(* IEC 61131-3 sources: RL_MAR/experiments/comparison/llm4plc/results/deepseek-ai-DeepSeek-V3.2_20260506_104945/20260506_111425, 4 files *)

(* ---- generated_code_iteration_0.st ---- *)
START_ST
FUNCTION_BLOCK TruckGarage
VAR_INPUT
    enter_flag : BOOL;
    exit_flag : BOOL;
    VehicleNumber_in : INT;
END_VAR
VAR_OUTPUT
    truck : T_TRUCK_INFO;
END_VAR
VAR_IN_OUT
    garage : ARRAY[1..3, 1..5] OF T_GARAGE_SLOT;
END_VAR
VAR
    state : INT; (* 0=IDLE, 1=ENTRY_ALLOCATION, 2=ENTRY_UPDATE, 3=EXIT_SEARCH, 4=EXIT_UPDATE *)
    prevState : INT;
    i : INT;
    j : INT;
    searchComplete : BOOL;
    vehicleFound : BOOL;
    tempVehicleNumber : INT;
    storedVehicleNumber : INT;
    enter_flag_prev : BOOL;
    exit_flag_prev : BOOL;
    enter_request : BOOL;
    exit_request : BOOL;
END_VAR

(* Edge detection for entry and exit flags *)
enter_request := enter_flag AND NOT enter_flag_prev;
exit_request := exit_flag AND NOT exit_flag_prev;
enter_flag_prev := enter_flag;
exit_flag_prev := exit_flag;

(* Main State Machine *)
CASE state OF
    0: (* IDLE *)
        (* Reset search indices based on next operation *)
        IF enter_request THEN
            state := 1;
            storedVehicleNumber := VehicleNumber_in;
            i := 3;
            j := 5;
            searchComplete := FALSE;
        ELSIF exit_request THEN
            state := 3;
            storedVehicleNumber := VehicleNumber_in;
            i := 1;
            j := 1;
            searchComplete := FALSE;
            vehicleFound := FALSE;
        END_IF;
        prevState := state;

    1: (* ENTRY_ALLOCATION *)
        IF NOT searchComplete THEN
            IF (i >= 1) AND (i <= 3) AND (j >= 1) AND (j <= 5) THEN
                IF NOT garage[i, j].Occupied THEN
                    state := 2; (* Free space found *)
                ELSE
                    (* Decrement column *)
                    j := j - 1;
                    IF j < 1 THEN
                        j := 5;
                        i := i - 1; (* Move to previous row *)
                    END_IF;
                    IF i < 1 THEN
                        searchComplete := TRUE; (* No space found *)
                    END_IF;
                END_IF;
            ELSE
                searchComplete := TRUE; (* Indices out of bounds *)
            END_IF;
        ELSE
            state := 0; (* No space found, return to IDLE *)
        END_IF;

    2: (* ENTRY_UPDATE *)
        garage[i, j].Occupied := TRUE;
        garage[i, j].VehicleNumber := storedVehicleNumber;
        state := 0;

    3: (* EXIT_SEARCH *)
        IF NOT searchComplete THEN
            IF (i >= 1) AND (i <= 3) AND (j >= 1) AND (j <= 5) THEN
                IF garage[i, j].Occupied AND (garage[i, j].VehicleNumber = storedVehicleNumber) THEN
                    vehicleFound := TRUE;
                    tempVehicleNumber := garage[i, j].VehicleNumber;
                    state := 4; (* Vehicle found *)
                ELSE
                    (* Increment column *)
                    j := j + 1;
                    IF j > 5 THEN
                        j := 1;
                        i := i + 1; (* Move to next row *)
                    END_IF;
                    IF i > 3 THEN
                        searchComplete := TRUE; (* Vehicle not found *)
                    END_IF;
                END_IF;
            ELSE
                searchComplete := TRUE; (* Indices out of bounds *)
            END_IF;
        ELSE
            state := 0; (* Vehicle not found, return to IDLE *)
        END_IF;

    4: (* EXIT_UPDATE *)
        garage[i, j].Occupied := FALSE;
        garage[i, j].VehicleNumber := 0;
        truck.row := i;
        truck.col := j;
        truck.VehicleNumber := tempVehicleNumber;
        state := 0;

END_CASE;

END_FUNCTION_BLOCK
END_ST

(* ---- generated_code_iteration_1.st ---- *)
START_REASON
The validation feedback indicates that the CODESYS compiler validation failed due to an "unknown type: 'T_TRUCK_INFO'". This error occurs because the data type `T_TRUCK_INFO` is used in the `VAR_OUTPUT` section but is not defined anywhere in the code. In Structured Text (ST) for CODESYS, all data types must be explicitly defined before they can be used. The original code likely assumed that `T_TRUCK_INFO` was predefined, but it is not. To fix this, I need to define the `T_TRUCK_INFO` structure. Additionally, the code uses `T_GARAGE_SLOT`, which is also undefined and must be defined. I will define both structures at the beginning of the code, before the `FUNCTION_BLOCK`, to ensure they are available for use. The structures should include the necessary fields: for `T_GARAGE_SLOT`, it should have `Occupied` (BOOL) and `VehicleNumber` (INT); for `T_TRUCK_INFO`, it should have `row` (INT), `col` (INT), and `VehicleNumber` (INT) based on the usage in the code. I will also ensure that the code adheres to the required formatting, such as using `END_VAR` correctly and maintaining the `FUNCTION_BLOCK` structure. No other errors were reported, so I will keep the existing logic intact while adding the missing type definitions.
END_REASON

START_ST
TYPE T_GARAGE_SLOT :
STRUCT
    Occupied : BOOL;
    VehicleNumber : INT;
END_STRUCT
END_TYPE

TYPE T_TRUCK_INFO :
STRUCT
    row : INT;
    col : INT;
    VehicleNumber : INT;
END_STRUCT
END_TYPE

FUNCTION_BLOCK TruckGarage
VAR_INPUT
    enter_flag : BOOL;
    exit_flag : BOOL;
    VehicleNumber_in : INT;
END_VAR
VAR_OUTPUT
    truck : T_TRUCK_INFO;
END_VAR
VAR_IN_OUT
    garage : ARRAY[1..3, 1..5] OF T_GARAGE_SLOT;
END_VAR
VAR
    state : INT; (* 0=IDLE, 1=ENTRY_ALLOCATION, 2=ENTRY_UPDATE, 3=EXIT_SEARCH, 4=EXIT_UPDATE *)
    prevState : INT;
    i : INT;
    j : INT;
    searchComplete : BOOL;
    vehicleFound : BOOL;
    tempVehicleNumber : INT;
    storedVehicleNumber : INT;
    enter_flag_prev : BOOL;
    exit_flag_prev : BOOL;
    enter_request : BOOL;
    exit_request : BOOL;
END_VAR

(* Edge detection for entry and exit flags *)
enter_request := enter_flag AND NOT enter_flag_prev;
exit_request := exit_flag AND NOT exit_flag_prev;
enter_flag_prev := enter_flag;
exit_flag_prev := exit_flag;

(* Main State Machine *)
CASE state OF
    0: (* IDLE *)
        (* Reset search indices based on next operation *)
        IF enter_request THEN
            state := 1;
            storedVehicleNumber := VehicleNumber_in;
            i := 3;
            j := 5;
            searchComplete := FALSE;
        ELSIF exit_request THEN
            state := 3;
            storedVehicleNumber := VehicleNumber_in;
            i := 1;
            j := 1;
            searchComplete := FALSE;
            vehicleFound := FALSE;
        END_IF;
        prevState := state;

    1: (* ENTRY_ALLOCATION *)
        IF NOT searchComplete THEN
            IF (i >= 1) AND (i <= 3) AND (j >= 1) AND (j <= 5) THEN
                IF NOT garage[i, j].Occupied THEN
                    state := 2; (* Free space found *)
                ELSE
                    (* Decrement column *)
                    j := j - 1;
                    IF j < 1 THEN
                        j := 5;
                        i := i - 1; (* Move to previous row *)
                    END_IF;
                    IF i < 1 THEN
                        searchComplete := TRUE; (* No space found *)
                    END_IF;
                END_IF;
            ELSE
                searchComplete := TRUE; (* Indices out of bounds *)
            END_IF;
        ELSE
            state := 0; (* No space found, return to IDLE *)
        END_IF;

    2: (* ENTRY_UPDATE *)
        garage[i, j].Occupied := TRUE;
        garage[i, j].VehicleNumber := storedVehicleNumber;
        state := 0;

    3: (* EXIT_SEARCH *)
        IF NOT searchComplete THEN
            IF (i >= 1) AND (i <= 3) AND (j >= 1) AND (j <= 5) THEN
                IF garage[i, j].Occupied AND (garage[i, j].VehicleNumber = storedVehicleNumber) THEN
                    vehicleFound := TRUE;
                    tempVehicleNumber := garage[i, j].VehicleNumber;
                    state := 4; (* Vehicle found *)
                ELSE
                    (* Increment column *)
                    j := j + 1;
                    IF j > 5 THEN
                        j := 1;
                        i := i + 1; (* Move to next row *)
                    END_IF;
                    IF i > 3 THEN
                        searchComplete := TRUE; (* Vehicle not found *)
                    END_IF;
                END_IF;
            ELSE
                searchComplete := TRUE; (* Indices out of bounds *)
            END_IF;
        ELSE
            state := 0; (* Vehicle not found, return to IDLE *)
        END_IF;

    4: (* EXIT_UPDATE *)
        garage[i, j].Occupied := FALSE;
        garage[i, j].VehicleNumber := 0;
        truck.row := i;
        truck.col := j;
        truck.VehicleNumber := tempVehicleNumber;
        state := 0;

END_CASE;

END_FUNCTION_BLOCK
END_ST

(* ---- generated_code_iteration_2.st ---- *)
START_REASON
The validation feedback indicates that the CODESYS compiler validation failed due to an "unknown type: 'T_TRUCK_INFO'" (in Chinese: "未知的类型: 'T_TRUCK_INFO'"). This error persists even after I added the TYPE definitions for both T_GARAGE_SLOT and T_TRUCK_INFO. The issue is likely that in CODESYS, TYPE definitions must be placed outside the FUNCTION_BLOCK, typically in a separate section or before the FUNCTION_BLOCK, but they must be properly scoped. In the previous code, I placed the TYPE definitions directly before the FUNCTION_BLOCK, but this might not be valid in all CODESYS contexts. Alternatively, the error might be because the TYPE definitions are not being recognized due to syntax or placement issues. I need to ensure the TYPE definitions are correctly formatted and placed. I will move the TYPE definitions to a separate section, ensuring they are properly closed with END_TYPE, and keep them before the FUNCTION_BLOCK. Additionally, I should verify that the STRUCT syntax is correct. No other errors were reported, so I will maintain the existing logic. I will also ensure that the code starts with START_ST and ends with END_ST as required.
END_REASON

START_ST
TYPE T_GARAGE_SLOT :
STRUCT
    Occupied : BOOL;
    VehicleNumber : INT;
END_STRUCT
END_TYPE

TYPE T_TRUCK_INFO :
STRUCT
    row : INT;
    col : INT;
    VehicleNumber : INT;
END_STRUCT
END_TYPE

FUNCTION_BLOCK TruckGarage
VAR_INPUT
    enter_flag : BOOL;
    exit_flag : BOOL;
    VehicleNumber_in : INT;
END_VAR
VAR_OUTPUT
    truck : T_TRUCK_INFO;
END_VAR
VAR_IN_OUT
    garage : ARRAY[1..3, 1..5] OF T_GARAGE_SLOT;
END_VAR
VAR
    state : INT; (* 0=IDLE, 1=ENTRY_ALLOCATION, 2=ENTRY_UPDATE, 3=EXIT_SEARCH, 4=EXIT_UPDATE *)
    prevState : INT;
    i : INT;
    j : INT;
    searchComplete : BOOL;
    vehicleFound : BOOL;
    tempVehicleNumber : INT;
    storedVehicleNumber : INT;
    enter_flag_prev : BOOL;
    exit_flag_prev : BOOL;
    enter_request : BOOL;
    exit_request : BOOL;
END_VAR

(* Edge detection for entry and exit flags *)
enter_request := enter_flag AND NOT enter_flag_prev;
exit_request := exit_flag AND NOT exit_flag_prev;
enter_flag_prev := enter_flag;
exit_flag_prev := exit_flag;

(* Main State Machine *)
CASE state OF
    0: (* IDLE *)
        (* Reset search indices based on next operation *)
        IF enter_request THEN
            state := 1;
            storedVehicleNumber := VehicleNumber_in;
            i := 3;
            j := 5;
            searchComplete := FALSE;
        ELSIF exit_request THEN
            state := 3;
            storedVehicleNumber := VehicleNumber_in;
            i := 1;
            j := 1;
            searchComplete := FALSE;
            vehicleFound := FALSE;
        END_IF;
        prevState := state;

    1: (* ENTRY_ALLOCATION *)
        IF NOT searchComplete THEN
            IF (i >= 1) AND (i <= 3) AND (j >= 1) AND (j <= 5) THEN
                IF NOT garage[i, j].Occupied THEN
                    state := 2; (* Free space found *)
                ELSE
                    (* Decrement column *)
                    j := j - 1;
                    IF j < 1 THEN
                        j := 5;
                        i := i - 1; (* Move to previous row *)
                    END_IF;
                    IF i < 1 THEN
                        searchComplete := TRUE; (* No space found *)
                    END_IF;
                END_IF;
            ELSE
                searchComplete := TRUE; (* Indices out of bounds *)
            END_IF;
        ELSE
            state := 0; (* No space found, return to IDLE *)
        END_IF;

    2: (* ENTRY_UPDATE *)
        garage[i, j].Occupied := TRUE;
        garage[i, j].VehicleNumber := storedVehicleNumber;
        state := 0;

    3: (* EXIT_SEARCH *)
        IF NOT searchComplete THEN
            IF (i >= 1) AND (i <= 3) AND (j >= 1) AND (j <= 5) THEN
                IF garage[i, j].Occupied AND (garage[i, j].VehicleNumber = storedVehicleNumber) THEN
                    vehicleFound := TRUE;
                    tempVehicleNumber := garage[i, j].VehicleNumber;
                    state := 4; (* Vehicle found *)
                ELSE
                    (* Increment column *)
                    j := j + 1;
                    IF j > 5 THEN
                        j := 1;
                        i := i + 1; (* Move to next row *)
                    END_IF;
                    IF i > 3 THEN
                        searchComplete := TRUE; (* Vehicle not found *)
                    END_IF;
                END_IF;
            ELSE
                searchComplete := TRUE; (* Indices out of bounds *)
            END_IF;
        ELSE
            state := 0; (* Vehicle not found, return to IDLE *)
        END_IF;

    4: (* EXIT_UPDATE *)
        garage[i, j].Occupied := FALSE;
        garage[i, j].VehicleNumber := 0;
        truck.row := i;
        truck.col := j;
        truck.VehicleNumber := tempVehicleNumber;
        state := 0;

END_CASE;

END_FUNCTION_BLOCK
END_ST

(* ---- generated_code_iteration_3.st ---- *)
START_REASON
The validation feedback indicates an encoding issue with the CODESYS compiler: "gbk codec can't decode byte 0xaa in position 149: illegal multibyte sequence". This suggests that there might be non-ASCII characters or special symbols in the code that the compiler cannot interpret correctly. Looking at the previous code, I notice that the comment "(* 0=IDLE, 1=ENTRY_ALLOCATION, 2=ENTRY_UPDATE, 3=EXIT_SEARCH, 4=EXIT_UPDATE *)" contains only ASCII characters, but there might be hidden or invisible characters introduced during copy-paste. The error occurs at position 149, which likely points to a specific character in the code. To fix this, I will rewrite the code from scratch, ensuring that all characters are standard ASCII and avoiding any special symbols. I will also ensure that the TYPE definitions are properly placed and that the code structure adheres to CODESYS standards. Additionally, I will simplify the comments to avoid any potential encoding issues. No functional changes are needed, but I will regenerate the code to eliminate any hidden characters.
END_REASON

START_ST
TYPE T_GARAGE_SLOT :
STRUCT
    Occupied : BOOL;
    VehicleNumber : INT;
END_STRUCT
END_TYPE

TYPE T_TRUCK_INFO :
STRUCT
    row : INT;
    col : INT;
    VehicleNumber : INT;
END_STRUCT
END_TYPE

FUNCTION_BLOCK TruckGarage
VAR_INPUT
    enter_flag : BOOL;
    exit_flag : BOOL;
    VehicleNumber_in : INT;
END_VAR
VAR_OUTPUT
    truck : T_TRUCK_INFO;
END_VAR
VAR_IN_OUT
    garage : ARRAY[1..3, 1..5] OF T_GARAGE_SLOT;
END_VAR
VAR
    state : INT;
    prevState : INT;
    i : INT;
    j : INT;
    searchComplete : BOOL;
    vehicleFound : BOOL;
    tempVehicleNumber : INT;
    storedVehicleNumber : INT;
    enter_flag_prev : BOOL;
    exit_flag_prev : BOOL;
    enter_request : BOOL;
    exit_request : BOOL;
END_VAR

enter_request := enter_flag AND NOT enter_flag_prev;
exit_request := exit_flag AND NOT exit_flag_prev;
enter_flag_prev := enter_flag;
exit_flag_prev := exit_flag;

CASE state OF
    0:
        IF enter_request THEN
            state := 1;
            storedVehicleNumber := VehicleNumber_in;
            i := 3;
            j := 5;
            searchComplete := FALSE;
        ELSIF exit_request THEN
            state := 3;
            storedVehicleNumber := VehicleNumber_in;
            i := 1;
            j := 1;
            searchComplete := FALSE;
            vehicleFound := FALSE;
        END_IF;
        prevState := state;

    1:
        IF NOT searchComplete THEN
            IF (i >= 1) AND (i <= 3) AND (j >= 1) AND (j <= 5) THEN
                IF NOT garage[i, j].Occupied THEN
                    state := 2;
                ELSE
                    j := j - 1;
                    IF j < 1 THEN
                        j := 5;
                        i := i - 1;
                    END_IF;
                    IF i < 1 THEN
                        searchComplete := TRUE;
                    END_IF;
                END_IF;
            ELSE
                searchComplete := TRUE;
            END_IF;
        ELSE
            state := 0;
        END_IF;

    2:
        garage[i, j].Occupied := TRUE;
        garage[i, j].VehicleNumber := storedVehicleNumber;
        state := 0;

    3:
        IF NOT searchComplete THEN
            IF (i >= 1) AND (i <= 3) AND (j >= 1) AND (j <= 5) THEN
                IF garage[i, j].Occupied AND (garage[i, j].VehicleNumber = storedVehicleNumber) THEN
                    vehicleFound := TRUE;
                    tempVehicleNumber := garage[i, j].VehicleNumber;
                    state := 4;
                ELSE
                    j := j + 1;
                    IF j > 5 THEN
                        j := 1;
                        i := i + 1;
                    END_IF;
                    IF i > 3 THEN
                        searchComplete := TRUE;
                    END_IF;
                END_IF;
            ELSE
                searchComplete := TRUE;
            END_IF;
        ELSE
            state := 0;
        END_IF;

    4:
        garage[i, j].Occupied := FALSE;
        garage[i, j].VehicleNumber := 0;
        truck.row := i;
        truck.col := j;
        truck.VehicleNumber := tempVehicleNumber;
        state := 0;

END_CASE;

END_FUNCTION_BLOCK
END_ST
